INTERFACE I_DS402GenericDrive

METHOD ExposedParameters
VAR_INPUT
	Enable : BOOL; 
    tRefreshDelay: TIME;
END_VAR
END_METHOD

METHOD Home
VAR_INPUT
END_VAR
END_METHOD

METHOD ModeOperation
VAR_INPUT
END_VAR
END_METHOD

METHOD MoveAbsolute
VAR_INPUT
END_VAR
END_METHOD

METHOD PersistParameters
VAR_INPUT
	 bEnable: BOOL;
END_VAR
END_METHOD

METHOD Power : BOOL
VAR_INPUT
END_VAR
END_METHOD

METHOD ReadDriveCodes : BOOL
END_METHOD

(*Read Piezo drive Motion parameters*)
METHOD ReadDriveParams : BOOL
VAR_INPUT
END_VAR
END_METHOD

METHOD Reset : BOOL
VAR_INPUT
END_VAR
END_METHOD

METHOD RestoreParameters
VAR_INPUT
END_VAR
END_METHOD

METHOD ScaleDriveParams
VAR_INPUT
END_VAR
END_METHOD

METHOD ScaleEncRawValue
VAR_INPUT
END_VAR
END_METHOD

METHOD ScaleHomeMotionParams
VAR_INPUT
END_VAR
END_METHOD

METHOD ScaleServoOffMotionParams
VAR_INPUT
END_VAR
END_METHOD

METHOD ScaleServoOnMotionParams : BOOL;
VAR_INPUT
END_VAR
END_METHOD

METHOD SetEnables
VAR_INPUT
END_VAR
END_METHOD

METHOD StateMachine
VAR_INPUT
END_VAR
END_METHOD

METHOD  StepMove
VAR_INPUT
	Enable : BOOL;
END_VAR
END_METHOD

METHOD UpdateDriveMonitoringParams
VAR_INPUT
    Enable : BOOL;
END_VAR
END_METHOD

METHOD UpdateEpicsStatus
VAR_INPUT
END_VAR
END_METHOD

METHOD UpdateServoOffMotionParams
VAR_INPUT
	Enable : BOOL;
END_VAR
END_METHOD

METHOD WriteParameterNC
VAR_INPUT
    Execute:BOOL;
    ParameterNumber : MC_AxisParameter;
    ParameterValue	: LREAL;
END_VAR
END_METHOD

END_INTERFACE

(* stored: Version 1.1.0.1
   Itf I_DS402GenericDrive: Id {49729736-8717-4a13-800f-a53162ccda84}
   Method ExposedParameters: Id {26e38a32-22d0-42ae-b0c6-5a30c1359c2c}
   Method Home: Id {f7b9941e-fd39-45a3-99c7-fc867c3625ba}
   Method ModeOperation: Id {6fb283a3-b1a1-4cbe-9046-2e4da66a2ed6}
   Method MoveAbsolute: Id {c32a9e13-f332-4841-9fc3-9751e2083446}
   Method PersistParameters: Id {2714254e-be9f-442a-9ff0-fec0cfde8ef7}
   Method Power: Id {08548eb9-8f7d-4758-8069-c44e4c6df0ba}
   Method ReadDriveCodes: Id {5baeecd3-c54d-4657-a7cc-e3729482e287}
   Method ReadDriveParams: Id {078b9a2c-2efa-40e1-9ad9-d1a70fc4b368}
   Method Reset: Id {43fc3192-2758-4d04-872e-08906cd5bf28}
   Method RestoreParameters: Id {b3ff829b-1562-4e27-8092-0b1cc927e533}
   Method ScaleDriveParams: Id {8ac3be16-28b8-4175-ae16-72a1e16261fb}
   Method ScaleEncRawValue: Id {5a3e0ac7-04c3-493b-9cb6-07a60972201e}
   Method ScaleHomeMotionParams: Id {2ab106ea-b09a-4819-bf0b-0e6b84eb1cf8}
   Method ScaleServoOffMotionParams: Id {b7054ca4-bda3-486f-9d59-a8ac6ece7055}
   Method ScaleServoOnMotionParams: Id {a2d7c6eb-36d7-439b-8657-67e88204b3ee}
   Method SetEnables: Id {b93a945e-5ba8-456d-9ebc-47294f36ee3e}
   Method StateMachine: Id {35531d1d-083e-4e0e-a309-4f04090b40cb}
   Method StepMove: Id {cdb17cc5-ff2a-49a3-bc83-37fe8e84d0f0}
   Method UpdateDriveMonitoringParams: Id {8610e279-04bc-4548-942d-f600acfb3079}
   Method UpdateEpicsStatus: Id {e22f0ab3-658b-45b7-b368-204fbd2d95fa}
   Method UpdateServoOffMotionParams: Id {1a1f77f3-ee6f-4689-a9b6-8149ebbedfec}
   Method WriteParameterNC: Id {3d85a3f6-b752-4960-b363-60741423f54d} *)
